FUNCTION_BLOCK DelayDoor
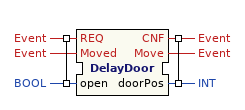
  EVENT_INPUT
    REQ WITH open;
    Moved;
  END_EVENT
  EVENT_OUTPUT
    CNF WITH doorPos;
    Move;
  END_EVENT
  VAR_INPUT
    open : BOOL;
  END_VAR
  VAR_OUTPUT
    doorPos : INT;
  END_VAR
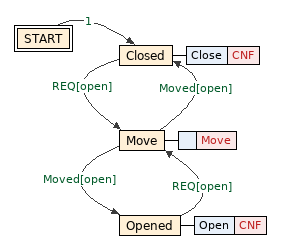
  EC_STATES
    START;
    Opened : Open -> CNF;
    Move : -> Move;
    Closed : Close -> CNF;
  END_STATES
  EC_TRANSITIONS
    Opened TO Move := REQ[open];
    Move TO Opened := Moved[open];
    START TO Closed := 1;
    Move TO Closed := Moved[open];
    Closed TO Move := REQ[open];
  END_TRANSITIONS
  ALGORITHM Open IN ST:
doorPos := 10;&#38;#10;
  END_ALGORITHM
  ALGORITHM Close IN ST:
doorPos := 0;&#38;#10;
  END_ALGORITHM
END_FUNCTION_BLOCK
